FUNCTION_BLOCK FB_HMI_Control
VAR_INPUT
	//iStationNumber : UINT;
	iRowNumber : UINT;
	
	iAdvanceLimit: BOOL;
	iReturnLimit: BOOL;
	iAdvanceCoil: BOOL;
	iReturnCoil: BOOL;
	
	iAdvanceTime:TIME;
	iReturnTime: TIME;
	
	iAdvanceInterlock: BOOL;
	iReturnInterlock: BOOL;

	iAdvancePrompt: BOOL;
	iReturnPrompt: BOOL;
	
	iConfig: WORD; //config for hide data
	
	iAdvanceNumber: UINT; //advance row number of sequence
	iReturnNumber: UINT; //return row number of sequence

	iUnits: STRING := ' mm';
	iPosn:   STRING := '0.0';
	iUsePV:BOOL :=FALSE; //TRUE to use process value (PV) from HMI row input 
END_VAR

VAR_OUTPUT
	qRow: UINT;
	qAdvanceReq: BOOL;
	qReturnReq: BOOL;
	qResultMessageOffset: UINT;
	qSP:STRING; //setpoint value returned from motionrow
END_VAR

VAR
	tNumMessagesPerRow: UINT;
	tMessageOffset: UINT;
	unitsString: STRING(255);
	
	advPulse:R_TRIG;
	retPulse:R_TRIG;
	
	
	strSPvalue:STRING;
	strPVvalue:STRING;
	strResultSPPVstring:STRING;
	
END_VAR

VAR_IN_OUT
	//NumRows: UINT;
	//MotionRowLocation: typeMotionRow;
	////MotionRowBtnLocation: typeMotionRowButtons;
	//iqMotionRecordStation: typeMotionRowArry;
	
	stndata:typeStation;
END_VAR

//theme:DrmpZtxr0kY

//calculate row order
qRow := iRowNumber * 20; //20 = number messages per row, or things per row

//Calculate number of rows
stndata.Data.NumOfRows := stndata.Data.NumOfRows + 1; //increment on scan of IN_OUT

//setup block clear down values
qAdvanceReq := FALSE;
qReturnReq := FALSE;
stndata.MotionRow[iRowNumber].Advance.Depth := FALSE;
stndata.MotionRow[iRowNumber].Returned.Depth := FALSE;
stndata.MotionRow[iRowNumber].Advance.RequestCoil := FALSE;
stndata.MotionRow[iRowNumber].Returned.RequestCoil := FALSE;
stndata.MotionRow[iRowNumber].Advance.InterlockOK := FALSE;
stndata.MotionRow[iRowNumber].Returned.InterlockOK := FALSE;
stndata.MotionRow[iRowNumber].Advance.Prompt := FALSE;
stndata.MotionRow[iRowNumber].Returned.Prompt := FALSE;
		

//advance feedback for HMI
IF stndata.MotionRowBtn[iRowNumber].btnAdvance	THEN	qAdvanceReq := TRUE;						END_IF
IF stndata.MotionRowBtn[iRowNumber].btnReturn	THEN	qReturnReq := TRUE;							END_IF

//limit switches
IF iAdvanceLimit					THEN	stndata.MotionRow[iRowNumber].Advance.Depth := TRUE;	END_IF
IF iReturnLimit						THEN	stndata.MotionRow[iRowNumber].Returned.Depth := TRUE;	END_IF

//coil feedback
IF iAdvanceCoil						THEN  	stndata.MotionRow[iRowNumber].Advance.RequestCoil := TRUE;	END_IF
IF iReturnCoil						THEN	stndata.MotionRow[iRowNumber].Returned.RequestCoil := TRUE; END_IF

//interlocks
IF iAdvanceInterlock AND (stndata.Data.Manual OR stndata.Data.SemiAuto)				THEN	stndata.MotionRow[iRowNumber].Advance.InterlockOK := TRUE;	END_IF
IF iReturnInterlock	 AND (stndata.Data.Manual OR stndata.Data.SemiAuto)				THEN	stndata.MotionRow[iRowNumber].Returned.InterlockOK := TRUE; END_IF

//prompts
IF iAdvancePrompt	AND (stndata.Data.Manual OR stndata.Data.SemiAuto)				THEN	stndata.MotionRow[iRowNumber].Advance.Prompt := TRUE;		END_IF
IF iReturnPrompt	AND (stndata.Data.Manual OR stndata.Data.SemiAuto)				THEN 	stndata.MotionRow[iRowNumber].Returned.Prompt := TRUE;		END_IF

//times
stndata.MotionRow[iRowNumber].Advance.TimeTaken		:= iAdvanceTime;
stndata.MotionRow[iRowNumber].Returned.TimeTaken	:= iReturnTime;

//Number of messages per motion, typ. 5 messages with space for more (10)
tNumMessagesPerRow						:= GlobalMessages.AllocMsgPerRow;

//define message position
//n= number of messages per row
tMessageOffset := tNumMessagesPerRow * iRowNumber;
qResultMessageOffset := tMessageOffset - tNumMessagesPerRow;

//config
//clear down config
stndata.MotionRow[iRowNumber].Advance.bHideButton		:= FALSE;
stndata.MotionRow[iRowNumber].Advance.bHideCoil			:= FALSE;
stndata.MotionRow[iRowNumber].Advance.bHideDepth		:= FALSE;
stndata.MotionRow[iRowNumber].Advance.bHideInterlock	:= FALSE;
stndata.MotionRow[iRowNumber].Advance.bHidePrompt		:= FALSE;
stndata.MotionRow[iRowNumber].Advance.bHideTime			:= FALSE;
stndata.MotionRow[iRowNumber].Returned.bHideButton		:= FALSE;
stndata.MotionRow[iRowNumber].Returned.bHideCoil		:= FALSE;
stndata.MotionRow[iRowNumber].Returned.bHideDepth		:= FALSE;
stndata.MotionRow[iRowNumber].Returned.bHideInterlock	:= FALSE;
stndata.MotionRow[iRowNumber].Returned.bHidePrompt		:= FALSE;
stndata.MotionRow[iRowNumber].Returned.bHideTime		:= FALSE;
stndata.MotionRow[iRowNumber].bHideName					:= FALSE;
stndata.MotionRow[iRowNumber].bHidePosn					:= FALSE;

//setup config
IF iConfig.0	THEN stndata.MotionRow[iRowNumber].Advance.bHideButton		:= TRUE; END_IF
IF iConfig.1	THEN stndata.MotionRow[iRowNumber].Advance.bHideCoil		:= TRUE; END_IF
IF iConfig.2	THEN stndata.MotionRow[iRowNumber].Advance.bHideDepth		:= TRUE; END_IF
IF iConfig.3	THEN stndata.MotionRow[iRowNumber].Advance.bHideInterlock	:= TRUE; END_IF
IF iConfig.4	THEN stndata.MotionRow[iRowNumber].Advance.bHidePrompt		:= TRUE; END_IF
IF iConfig.5	THEN stndata.MotionRow[iRowNumber].Advance.bHideTime		:= TRUE; END_IF
IF iConfig.6	THEN stndata.MotionRow[iRowNumber].Returned.bHideButton		:= TRUE; END_IF
IF iConfig.7	THEN stndata.MotionRow[iRowNumber].Returned.bHideCoil		:= TRUE; END_IF
IF iConfig.8	THEN stndata.MotionRow[iRowNumber].Returned.bHideDepth		:= TRUE; END_IF
IF iConfig.9	THEN stndata.MotionRow[iRowNumber].Returned.bHideInterlock	:= TRUE; END_IF
IF iConfig.10	THEN stndata.MotionRow[iRowNumber].Returned.bHidePrompt		:= TRUE; END_IF
IF iConfig.11	THEN stndata.MotionRow[iRowNumber].Returned.bHideTime		:= TRUE; END_IF
IF iConfig.12	THEN stndata.MotionRow[iRowNumber].bHidePosn				:= TRUE; END_IF
IF iConfig.13	THEN stndata.MotionRow[iRowNumber].bHideName				:= TRUE; END_IF


//advance number of order
stndata.MotionRow[iRowNumber].Advance.NumberOrder := iAdvanceNumber;
//return number of order
stndata.MotionRow[iRowNumber].Returned.NumberOrder := iReturnNumber;

IF iUsePV THEN
	
	//assemble SP / PV text
	//SP: 123.456 PV:321.654 mm 
	stndata.MotionRow[iRowNumber].strPosn := CONCAT(STR1:=iPosn, STR2:=iUnits);
	
	strSPvalue := CONCAT(STR1:='SP: ', STR2:=stndata.MotionRowBtn[iRowNumber].stnPosnInput);
	strPVvalue := CONCAT(STR1:='PV: ', STR2:=stndata.MotionRow[iRowNumber].strPosn);	
	strPVvalue := CONCAT(STR1:=' / ', STR2:=strPVvalue);	
	strResultSPPVstring := CONCAT(STR1:=strSPvalue, STR2:=strPVvalue);
	
	stndata.MotionRow[iRowNumber].strPosn := strResultSPPVstring;
	qSP := stndata.MotionRowBtn[iRowNumber].stnPosnInput;
	 ELSE
	//assemble posn string
	// xxx.xxx <units>
	// 123.456 mm
	stndata.MotionRow[iRowNumber].strPosn := CONCAT(STR1:=iPosn, STR2:=iUnits);
	qSP := '0.0';
	
END_IF

IF gHMIButtons.btnAbsMode THEN
	stndata.MotionRow[iRowNumber].bIsAbsSymSwitch := TRUE;
	ELSE
	stndata.MotionRow[iRowNumber].bIsAbsSymSwitch := FALSE;
END_IF

//setup default colour
stndata.MotionRow[iRowNumber].Advance.CoilColour	:= HMIColour.colourGreyBackground;
stndata.MotionRow[iRowNumber].Returned.CoilColour	:= HMIColour.colourGreyBackground;
stndata.MotionRow[iRowNumber].Advance.FdbkColour	:= HMIColour.colourGreyBackground;
stndata.MotionRow[iRowNumber].Returned.FdbkColour	:= HMIColour.colourGreyBackground;
	
//colour setup for row
IF	iAdvanceCoil		THEN stndata.MotionRow[iRowNumber].Advance.CoilColour	:= HMIColour.colourGreen;	END_IF
IF	iReturnCoil		THEN stndata.MotionRow[iRowNumber].Returned.CoilColour	:= HMIColour.colourYellow;	END_IF
IF	iAdvanceLimit	THEN stndata.MotionRow[iRowNumber].Advance.FdbkColour	:= HMIColour.colourGreen;	END_IF
IF	iReturnLimit	THEN stndata.MotionRow[iRowNumber].Returned.FdbkColour	:= HMIColour.colourYellow;	END_IF

//record number of motions
actUpdateRecord();

ACTION actUpdateRecord:
//generate pulse per motion limit
advPulse(CLK:=iAdvanceLimit);
retPulse(CLK:=iReturnLimit);


//update motion record
IF advPulse.Q THEN
		stndata.MotionRecordStation.data[iRowNumber].Advanced 
	:=	stndata.MotionRecordStation.data[iRowNumber].Advanced  + 1;
END_IF

//update motion record
IF retPulse.Q THEN
		stndata.MotionRecordStation.data[iRowNumber].Returned 
	:=	stndata.MotionRecordStation.data[iRowNumber].Returned + 1;
END_IF
END_ACTION

END_FUNCTION_BLOCK

(* stored: Version 1.1.0.1, ProductVersion 3.1.4024.11
   POU FB_HMI_Control: Id {01ed13c7-6a6a-43a8-8dee-d4708dd83b55}, SpecialFunc None
   Action actUpdateRecord: Id {434e14d4-429c-464f-877e-d0874076e223} *)
